(* CoDeSys 2.3 export: AUTO_CARRITOS.EXP *)

(* POU Automatico/Exterior/Control_AGV/Auto_Carritos, LD *)
PROGRAM Auto_Carritos
VAR
	Carrito_1: Control_carritos;
	Carrito_2: Control_carritos;
	Espera1: BOOL;
	Espera2: BOOL;
	Temp_Carrito: TON;
	FT2: BOOL;
	AT2: BOOL;
END_VAR
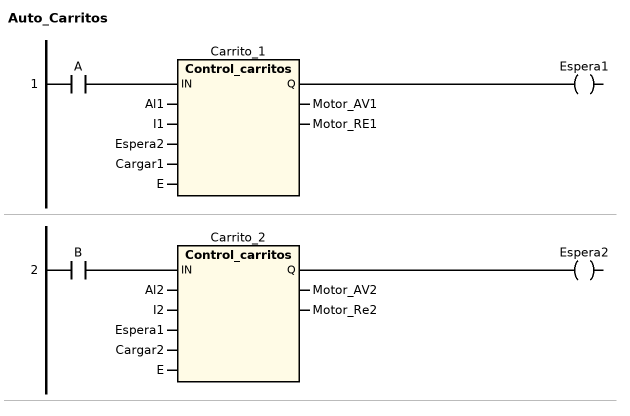
_LD_ (* Ladder Diagram *)
NETWORK 1
	[A] - Carrito_1:Control_carritos(*, Al1, I1, Espera2, Cargar1, E, out 2 => Motor_AV1, out 3 => Motor_RE1) --- (Espera1)
NETWORK 2
	[B] - Carrito_2:Control_carritos(*, Al2, I2, Espera1, Cargar2, E, out 2 => Motor_AV2, out 3 => Motor_Re2) --- (Espera2)
_END_LD_
END_PROGRAM
